      ;FOLD -- Start StartAcknowledge AUS -- ;%{SE}%MKUKATPVW %CVW_COM %VCOMMENT %P 2:-- Start StartAcknowledge AUS --, 3: VW_COMMENT
      ;ENDFOLD
      ;FOLD A3512 = AUS ;%{SE}%MKUKATPVW %CVW_SPS %VBOASG %P 2:A3512 = AUS, 3: BOASG
         $OUT[3512] = FALSE
      ;ENDFOLD
      ;FOLD -- RSK Fehlerausgabe Kraftaufbau -- ;%{SE}%MKUKATPVW %CVW_COM %VCOMMENT %P 2:-- RSK Fehlerausgabe Kraftaufbau --, 3: VW_COMMENT
      ;ENDFOLD
      ;FOLD F325 = EIN ;%{SE}%MKUKATPVW %CVW_SPS %VBOASG %P 2:F325 = EIN, 3: BOASG
         $FLAG[325] = TRUE
      ;ENDFOLD
      ;FOLD -- RSK Fehlerausgabe -- ;%{SE}%MKUKATPVW %CVW_COM %VCOMMENT %P 2:-- RSK Fehlerausgabe --, 3: VW_COMMENT
      ;ENDFOLD
      ;FOLD F327 = EIN ;%{SE}%MKUKATPVW %CVW_SPS %VBOASG %P 2:F327 = EIN, 3: BOASG
         $FLAG[327] = TRUE
      ;ENDFOLD
      ;FOLD F174 = !F327 & F174 ;%{SE}%MKUKATPVW %CVW_SPS %VBOASG %P 2:F174 = !F327 & F174, 3: BOASG
         $FLAG[174] = NOT $FLAG[327] AND $FLAG[174]
      ;ENDFOLD
      ;FOLD F175 = F327 + F175 ;%{SE}%MKUKATPVW %CVW_SPS %VBOASG %P 2:F175 = F327 + F175, 3: BOASG
         $FLAG[175] = $FLAG[327] OR $FLAG[175]
      ;ENDFOLD
      ;FOLD -- RSK Sammelstoerung -- ;%{SE}%MKUKATPVW %CVW_COM %VCOMMENT %P 2:-- RSK Sammelstoerung --, 3: VW_COMMENT
      ;ENDFOLD
      ;FOLD F329 = F325 + F326 + F327 ;%{SE}%MKUKATPVW %CVW_SPS %VBOASG %P 2:F329 = F325 + F326 + F327, 3: BOASG
         $FLAG[329] = $FLAG[325] OR $FLAG[326] OR $FLAG[327]
      ;ENDFOLD
      ;FOLD A3519 = EIN ;%{SE}%MKUKATPVW %CVW_SPS %VBOASG %P 2:A3519 = EIN, 3: BOASG
         $OUT[3519] = TRUE
      ;ENDFOLD
      ;FOLD -- Flagbildung Wiederholfraesen -- ;%{SE}%MKUKATPVW %CVW_COM %VCOMMENT %P 2:-- Flagbildung Wiederholfraesen --, 3: VW_COMMENT
      ;ENDFOLD
      ;FOLD F749 = F329 & !A3518 ;%{SE}%MKUKATPVW %CVW_SPS %VBOASG %P 2:F749 = F329 & !A3518, 3: BOASG
         $FLAG[749] = $FLAG[329] AND NOT $OUT[3518]
      ;ENDFOLD
      ;FOLD A204 = A3518 ;%{SE}%MKUKATPVW %CVW_SPS %VBOASG %P 2:A204 = A3518, 3: BOASG
         $OUT[204] = $OUT[3518]
      ;ENDFOLD
      ;FOLD Schritt 303 = A3926 & A3518 & (E26 + E27) ;%{SE}%MKUKATPVW %CVW_SPS %VST_CON %P 2:Schritt 303 = A3926 & A3518 & (E26 + E27), 3: ST_CON
         IF $OUT[3926] AND $OUT[3518] AND ($IN[26] OR $IN[27]) THEN
            PREV_STEP[9] = APP_INT_STEP[9]
            APP_INT_STEP[9] = 303
         ENDIF
      ;ENDFOLD
      ;FOLD Schritt 303 = A3926 & !A3518 & F749 & A4039 ;%{SE}%MKUKATPVW %CVW_SPS %VST_CON %P 2:Schritt 303 = A3926 & !A3518 & F749 & A4039, 3: ST_CON
         IF $OUT[3926] AND NOT $OUT[3518] AND $FLAG[749] AND $OUT[4039] THEN
            PREV_STEP[9] = APP_INT_STEP[9]
            APP_INT_STEP[9] = 303
         ENDIF
      ;ENDFOLD
   ;ENDFOLD
   ;FOLD SCHRITT 333 -- st. RZ3 # Acknowledge -- ;%{P}%MKUKATPVW,%CSTEP,%VST_NR,%P 1:SCHRITT, 2:333, 3: st. RZ3 # Acknowledge
      ;FOLD ;%{H}
         Case 333
      ;ENDFOLD
      ;FOLD -- ServoGun SZ1 oeffnen -- ;%{SE}%MKUKATPVW %CVW_COM %VCOMMENT %P 2:-- ServoGun SZ1 oeffnen --, 3: VW_COMMENT
      ;ENDFOLD
      ;FOLD A3511 = AUS ;%{SE}%MKUKATPVW %CVW_SPS %VBOASG %P 2:A3511 = AUS, 3: BOASG
         $OUT[3511] = FALSE
      ;ENDFOLD
      ;FOLD A3512 = EIN ;%{SE}%MKUKATPVW %CVW_SPS %VBOASG %P 2:A3512 = EIN, 3: BOASG
         $OUT[3512] = TRUE
      ;ENDFOLD
      ;FOLD -- RSK Fehlerausgabe Kraftaufbau -- ;%{SE}%MKUKATPVW %CVW_COM %VCOMMENT %P 2:-- RSK Fehlerausgabe Kraftaufbau --, 3: VW_COMMENT
      ;ENDFOLD
      ;FOLD F325 = AUS ;%{SE}%MKUKATPVW %CVW_SPS %VBOASG %P 2:F325 = AUS, 3: BOASG
         $FLAG[325] = FALSE
      ;ENDFOLD
      ;FOLD -- RSK Fehlerausgabe -- ;%{SE}%MKUKATPVW %CVW_COM %VCOMMENT %P 2:-- RSK Fehlerausgabe --, 3: VW_COMMENT
      ;ENDFOLD
      ;FOLD F327 = AUS ;%{SE}%MKUKATPVW %CVW_SPS %VBOASG %P 2:F327 = AUS, 3: BOASG
         $FLAG[327] = FALSE
      ;ENDFOLD
      ;FOLD -- RSK Fehlerausgabe -- ;%{SE}%MKUKATPVW %CVW_COM %VCOMMENT %P 2:-- RSK Fehlerausgabe --, 3: VW_COMMENT
      ;ENDFOLD
      ;FOLD F329 = AUS ;%{SE}%MKUKATPVW %CVW_SPS %VBOASG %P 2:F329 = AUS, 3: BOASG
         $FLAG[329] = FALSE
      ;ENDFOLD
      ;FOLD Schritt 334 = A3926 & A3506 & A3505 & !A3507 & A4039 ;%{SE}%MKUKATPVW %CVW_SPS %VST_CON %P 2:Schritt 334 = A3926 & A3506 & A3505 & !A3507 & A4039, 3: ST_CON
         IF $OUT[3926] AND $OUT[3506] AND $OUT[3505] AND NOT $OUT[3507] AND $OUT[4039] THEN
            PREV_STEP[9] = APP_INT_STEP[9]
            APP_INT_STEP[9] = 334
         ENDIF
      ;ENDFOLD
   ;ENDFOLD
   ;FOLD SCHRITT 334 -- st. RZ3 # Ende -- ;%{P}%MKUKATPVW,%CSTEP,%VST_NR,%P 1:SCHRITT, 2:334, 3: st. RZ3 # Ende
      ;FOLD ;%{H}
         Case 334
      ;ENDFOLD
      ;FOLD -- Hilfsflag SK Programmwechsel -- ;%{SE}%MKUKATPVW %CVW_COM %VCOMMENT %P 2:-- Hilfsflag SK Programmwechsel --, 3: VW_COMMENT
      ;ENDFOLD
      ;FOLD F334 = AUS ;%{SE}%MKUKATPVW %CVW_SPS %VBOASG %P 2:F334 = AUS, 3: BOASG
         $FLAG[334] = FALSE
      ;ENDFOLD
      ;FOLD A116 = AUS ;%{SE}%MKUKATPVW %CVW_SPS %VBOASG %P 2:A116 = AUS, 3: BOASG
         $OUT[116] = FALSE
      ;ENDFOLD
      ;FOLD A192 = AUS ;%{SE}%MKUKATPVW %CVW_SPS %VBOASG %P 2:A192 = AUS, 3: BOASG
         $OUT[192] = FALSE
      ;ENDFOLD
      ;FOLD A1107 = AUS ;%{SE}%MKUKATPVW %CVW_SPS %VBOASG %P 2:A1107 = AUS, 3: BOASG
         $OUT[1107] = FALSE
      ;ENDFOLD
      ;FOLD A3518 = AUS ;%{SE}%MKUKATPVW %CVW_SPS %VBOASG %P 2:A3518 = AUS, 3: BOASG
         $OUT[3518] = FALSE
      ;ENDFOLD
      ;FOLD A3519 = AUS ;%{SE}%MKUKATPVW %CVW_SPS %VBOASG %P 2:A3519 = AUS, 3: BOASG
         $OUT[3519] = FALSE
      ;ENDFOLD
      ;FOLD F836 = AUS ;%{SE}%MKUKATPVW %CVW_SPS %VBOASG %P 2:F836 = AUS, 3: BOASG
         $FLAG[836] = FALSE
      ;ENDFOLD
      ;FOLD -- Start Init Same AUS -- ;%{SE}%MKUKATPVW %CVW_COM %VCOMMENT %P 2:-- Start Init Same AUS --, 3: VW_COMMENT
      ;ENDFOLD
      ;FOLD A3514 = AUS ;%{SE}%MKUKATPVW %CVW_SPS %VBOASG %P 2:A3514 = AUS, 3: BOASG
         $OUT[3514] = FALSE
      ;ENDFOLD
      ;FOLD -- Start Spot AUS -- ;%{SE}%MKUKATPVW %CVW_COM %VCOMMENT %P 2:-- Start Spot AUS --, 3: VW_COMMENT
      ;ENDFOLD
      ;FOLD A3511 = AUS ;%{SE}%MKUKATPVW %CVW_SPS %VBOASG %P 2:A3511 = AUS, 3: BOASG
         $OUT[3511] = FALSE
      ;ENDFOLD
      ;FOLD -- Start Dress AUS -- ;%{SE}%MKUKATPVW %CVW_COM %VCOMMENT %P 2:-- Start Dress AUS --, 3: VW_COMMENT
      ;ENDFOLD
      ;FOLD A3510 = AUS ;%{SE}%MKUKATPVW %CVW_SPS %VBOASG %P 2:A3510 = AUS, 3: BOASG
         $OUT[3510] = FALSE
      ;ENDFOLD
      ;FOLD -- Start Init New AUS -- ;%{SE}%MKUKATPVW %CVW_COM %VCOMMENT %P 2:-- Start Init New AUS --, 3: VW_COMMENT
      ;ENDFOLD
      ;FOLD A3513 = AUS ;%{SE}%MKUKATPVW %CVW_SPS %VBOASG %P 2:A3513 = AUS, 3: BOASG
         $OUT[3513] = FALSE
      ;ENDFOLD
      ;FOLD -- Dress in Position AUS -- ;%{SE}%MKUKATPVW %CVW_COM %VCOMMENT %P 2:-- Dress in Position AUS --, 3: VW_COMMENT
      ;ENDFOLD
      ;FOLD A3935 = AUS ;%{SE}%MKUKATPVW %CVW_SPS %VBOASG %P 2:A3935 = AUS, 3: BOASG
         $OUT[3935] = FALSE
      ;ENDFOLD
      ;FOLD -- Dress Fin AUS -- ;%{SE}%MKUKATPVW %CVW_COM %VCOMMENT %P 2:-- Dress Fin AUS --, 3: VW_COMMENT
      ;ENDFOLD
      ;FOLD A3936 = AUS ;%{SE}%MKUKATPVW %CVW_SPS %VBOASG %P 2:A3936 = AUS, 3: BOASG
         $OUT[3936] = FALSE
      ;ENDFOLD
      ;FOLD -- Start StartAcknowledge AUS -- ;%{SE}%MKUKATPVW %CVW_COM %VCOMMENT %P 2:-- Start StartAcknowledge AUS --, 3: VW_COMMENT
      ;ENDFOLD
      ;FOLD A3512 = AUS ;%{SE}%MKUKATPVW %CVW_SPS %VBOASG %P 2:A3512 = AUS, 3: BOASG
         $OUT[3512] = FALSE
      ;ENDFOLD
      ;FOLD -- RSK Sammelstoerung -- ;%{SE}%MKUKATPVW %CVW_COM %VCOMMENT %P 2:-- RSK Sammelstoerung --, 3: VW_COMMENT
      ;ENDFOLD
      ;FOLD F329 = F196 ;%{SE}%MKUKATPVW %CVW_SPS %VBOASG %P 2:F329 = F196, 3: BOASG
         $FLAG[329] = $FLAG[196]
      ;ENDFOLD
      ;FOLD F185 = (!E1106 & E787 & !E1108 & !F830) + F196 & (E26 + E27) ;%{SE}%MKUKATPVW %CVW_SPS %VBOASG %P 2:F185 = (!E1106 & E787 & !E1108 & !F830) + F196 & (E26 + E27), 3: BOASG
         $FLAG[185] = (NOT $IN[1106] AND $IN[787] AND NOT $IN[1108] AND NOT $FLAG[830]) OR $FLAG[196] AND ($IN[26] OR $IN[27])
      ;ENDFOLD
      ;FOLD SCHRITT 1 = F185 & A4039 & A3926 & A3506 & A3505 ;%{SE}%MKUKATPVW %CVW_SPS %VST_CON %P 2:SCHRITT 1 = F185 & A4039 & A3926 & A3506 & A3505, 3: ST_CON
         IF $FLAG[185] AND $OUT[4039] AND $OUT[3926] AND $OUT[3506] AND $OUT[3505] THEN
            PREV_STEP[9] = APP_INT_STEP[9]
            APP_INT_STEP[9] = 1
         ENDIF
      ;ENDFOLD
   ;ENDFOLD
   ;FOLD SCHRITT 350 -- st. RZ3 # Fehler SGB -- ;%{P}%MKUKATPVW,%CSTEP,%VST_NR,%P 1:SCHRITT, 2:350, 3: st. RZ3 # Fehler SGB
      ;FOLD ;%{H}
         Case 350
      ;ENDFOLD
      ;FOLD -- Start Init Same AUS -- ;%{SE}%MKUKATPVW %CVW_COM %VCOMMENT %P 2:-- Start Init Same AUS --, 3: VW_COMMENT
      ;ENDFOLD
      ;FOLD A3514 = AUS ;%{SE}%MKUKATPVW %CVW_SPS %VBOASG %P 2:A3514 = AUS, 3: BOASG
         $OUT[3514] = FALSE
      ;ENDFOLD
      ;FOLD -- Start Spot AUS -- ;%{SE}%MKUKATPVW %CVW_COM %VCOMMENT %P 2:-- Start Spot AUS --, 3: VW_COMMENT
      ;ENDFOLD
      ;FOLD A3511 = AUS ;%{SE}%MKUKATPVW %CVW_SPS %VBOASG %P 2:A3511 = AUS, 3: BOASG
         $OUT[3511] = FALSE
      ;ENDFOLD
      ;FOLD -- Start Dress AUS -- ;%{SE}%MKUKATPVW %CVW_COM %VCOMMENT %P 2:-- Start Dress AUS --, 3: VW_COMMENT
      ;ENDFOLD
      ;FOLD A3510 = AUS ;%{SE}%MKUKATPVW %CVW_SPS %VBOASG %P 2:A3510 = AUS, 3: BOASG
         $OUT[3510] = FALSE
      ;ENDFOLD
      ;FOLD -- Start Init New AUS -- ;%{SE}%MKUKATPVW %CVW_COM %VCOMMENT %P 2:-- Start Init New AUS --, 3: VW_COMMENT
      ;ENDFOLD
      ;FOLD A3513 = AUS ;%{SE}%MKUKATPVW %CVW_SPS %VBOASG %P 2:A3513 = AUS, 3: BOASG
         $OUT[3513] = FALSE
      ;ENDFOLD
      ;FOLD -- Start Dress in Position AUS -- ;%{SE}%MKUKATPVW %CVW_COM %VCOMMENT %P 2:-- Start Dress in Position AUS --, 3: VW_COMMENT
      ;ENDFOLD
      ;FOLD A3935 = AUS ;%{SE}%MKUKATPVW %CVW_SPS %VBOASG %P 2:A3935 = AUS, 3: BOASG
         $OUT[3935] = FALSE
      ;ENDFOLD
      ;FOLD -- Start Dress Fin AUS -- ;%{SE}%MKUKATPVW %CVW_COM %VCOMMENT %P 2:-- Start Dress Fin AUS --, 3: VW_COMMENT
      ;ENDFOLD
      ;FOLD A3936 = AUS ;%{SE}%MKUKATPVW %CVW_SPS %VBOASG %P 2:A3936 = AUS, 3: BOASG
         $OUT[3936] = FALSE
      ;ENDFOLD
      ;FOLD -- Start StartAcknowledge EIN -- ;%{SE}%MKUKATPVW %CVW_COM %VCOMMENT %P 2:-- Start StartAcknowledge EIN --, 3: VW_COMMENT
      ;ENDFOLD
      ;FOLD A3512 = EIN ;%{SE}%MKUKATPVW %CVW_SPS %VBOASG %P 2:A3512 = EIN, 3: BOASG
         $OUT[3512] = TRUE
      ;ENDFOLD
      ;FOLD -- Kommentar -- ;%{SE}%MKUKATPVW %CVW_COM %VCOMMENT %P 2:-- Kommentar --, 3: VW_COMMENT
      ;ENDFOLD
      ;FOLD Schritt 351 = A4039 & A140 & !A3507 & A3506 & A3505 ;%{SE}%MKUKATPVW %CVW_SPS %VST_CON %P 2:Schritt 351 = A4039 & A140 & !A3507 & A3506 & A3505, 3: ST_CON
         IF $OUT[4039] AND $OUT[140] AND NOT $OUT[3507] AND $OUT[3506] AND $OUT[3505] THEN
            PREV_STEP[9] = APP_INT_STEP[9]
            APP_INT_STEP[9] = 351
         ENDIF
      ;ENDFOLD
   ;ENDFOLD
   ;FOLD SCHRITT 351 -- st. RZ3 # Fehler SGB -- ;%{P}%MKUKATPVW,%CSTEP,%VST_NR,%P 1:SCHRITT, 2:351, 3: st. RZ3 # Fehler SGB
      ;FOLD ;%{H}
         Case 351
      ;ENDFOLD
      ;FOLD -- Start StartAcknowledge AUS -- ;%{SE}%MKUKATPVW %CVW_COM %VCOMMENT %P 2:-- Start StartAcknowledge AUS --, 3: VW_COMMENT
      ;ENDFOLD
      ;FOLD A3512 = AUS ;%{SE}%MKUKATPVW %CVW_SPS %VBOASG %P 2:A3512 = AUS, 3: BOASG
         $OUT[3512] = FALSE
      ;ENDFOLD
      ;FOLD SCHRITT 1 = A4039 & A204 ;%{SE}%MKUKATPVW %CVW_SPS %VST_CON %P 2:SCHRITT 1 = A4039 & A204, 3: ST_CON
         IF $OUT[4039] AND $OUT[204] THEN
            PREV_STEP[9] = APP_INT_STEP[9]
            APP_INT_STEP[9] = 1
         ENDIF
      ;ENDFOLD
   ;ENDFOLD
   ;FOLD SCHRITT 390 -- st. RZ3 Setzhub 2 -- ;%{P}%MKUKATPVW,%CSTEP,%VST_NR,%P 1:SCHRITT, 2:390, 3: st. RZ3 Setzhub 2
      ;FOLD ;%{H}
         Case 390
      ;ENDFOLD
      ;FOLD -- Druckvorgabe SK1/ServoGun -- ;%{SE}%MKUKATPVW %CVW_COM %VCOMMENT %P 2:-- Druckvorgabe SK1/ServoGun --, 3: VW_COMMENT
      ;ENDFOLD
      ;FOLD bin7 ( F174 ) = 61 ;%{SE}%MKUKATPVW %CVW_SPS %VARIASG %P 2:bin7 ( F174 ) = 61, 3: ARIASG
         VW(#BINOUT,$FLAG[174],7,61)
      ;ENDFOLD
      ;FOLD bin31 ( F174 ) = 61 ;%{SE}%MKUKATPVW %CVW_SPS %VARIASG %P 2:bin31 ( F174 ) = 61, 3: ARIASG
         VW(#BINOUT,$FLAG[174],31,61)
      ;ENDFOLD
      ;FOLD -- Wartezeit Programmwechsel SK -- ;%{SE}%MKUKATPVW %CVW_COM %VCOMMENT %P 2:-- Wartezeit Programmwechsel SK --, 3: VW_COMMENT
      ;ENDFOLD
      ;FOLD T8 ( !F334 ) = -2[1/10Sek] ;%{SE}%MKUKATPVW %CVW_SPS %VTASG %P 2:T8 ( !F334 ) = -2[1/10Sek], 3: TASG
         VW(#SET_TIME,NOT $FLAG[334],8,0,-2)
      ;ENDFOLD
      ;FOLD -- Ueberwachungszeit ServoGun Setzhub 2 -- ;%{SE}%MKUKATPVW %CVW_COM %VCOMMENT %P 2:-- Ueberwachungszeit ServoGun Setzhub 2 --, 3: VW_COMMENT
      ;ENDFOLD
      ;FOLD t9 ( EIN ) = -80[1/10Sek] ;%{SE}%MKUKATPVW %CVW_SPS %VTASG %P 2:t9 ( EIN ) = -80[1/10Sek], 3: TASG
         VW(#SET_TIME,TRUE,9,0,-80)
      ;ENDFOLD
      ;FOLD -- Hilfsflag SK Programmwechsel -- ;%{SE}%MKUKATPVW %CVW_COM %VCOMMENT %P 2:-- Hilfsflag SK Programmwechsel --, 3: VW_COMMENT
      ;ENDFOLD
      ;FOLD F334 = EIN ;%{SE}%MKUKATPVW %CVW_SPS %VBOASG %P 2:F334 = EIN, 3: BOASG
         $FLAG[334] = TRUE
      ;ENDFOLD
      ;FOLD A3512 = AUS ;%{SE}%MKUKATPVW %CVW_SPS %VBOASG %P 2:A3512 = AUS, 3: BOASG
         $OUT[3512] = FALSE
      ;ENDFOLD
      ;FOLD Schritt 391 = T8 & A4039 & A3506 & A3505 & !A3507 ;%{SE}%MKUKATPVW %CVW_SPS %VST_CON %P 2:Schritt 391 = T8 & A4039 & A3506 & A3505 & !A3507, 3: ST_CON
         IF $TIMER_FLAG[8] AND $OUT[4039] AND $OUT[3506] AND $OUT[3505] AND NOT $OUT[3507] THEN
            PREV_STEP[9] = APP_INT_STEP[9]
            APP_INT_STEP[9] = 391
         ENDIF
      ;ENDFOLD
   ;ENDFOLD
   ;FOLD SCHRITT 391 -- st. RZ3 Setzhub 2 # InitSame -- ;%{P}%MKUKATPVW,%CSTEP,%VST_NR,%P 1:SCHRITT, 2:391, 3: st. RZ3 Setzhub 2 # InitSame
      ;FOLD ;%{H}
         Case 391
      ;ENDFOLD
      ;FOLD -- Hilfsflag SK Programmwechsel -- ;%{SE}%MKUKATPVW %CVW_COM %VCOMMENT %P 2:-- Hilfsflag SK Programmwechsel --, 3: VW_COMMENT
      ;ENDFOLD
      ;FOLD F334 = AUS ;%{SE}%MKUKATPVW %CVW_SPS %VBOASG %P 2:F334 = AUS, 3: BOASG
         $FLAG[334] = FALSE
      ;ENDFOLD
      ;FOLD -- Zeit fuer Setzhub -- ;%{SE}%MKUKATPVW %CVW_COM %VCOMMENT %P 2:-- Zeit fuer Setzhub --, 3: VW_COMMENT
      ;ENDFOLD
      ;FOLD T8 ( EIN ) = -80[1/10Sek] ;%{SE}%MKUKATPVW %CVW_SPS %VTASG %P 2:T8 ( EIN ) = -80[1/10Sek], 3: TASG
         VW(#SET_TIME,TRUE,8,0,-80)
      ;ENDFOLD
      ;FOLD -- Messen nach Fraesen -- ;%{SE}%MKUKATPVW %CVW_COM %VCOMMENT %P 2:-- Messen nach Fraesen --, 3: VW_COMMENT
      ;ENDFOLD
      ;FOLD A3514 = EIN ;%{SE}%MKUKATPVW %CVW_SPS %VBOASG %P 2:A3514 = EIN, 3: BOASG
         $OUT[3514] = TRUE
      ;ENDFOLD
      ;FOLD A3510 = EIN ;%{SE}%MKUKATPVW %CVW_SPS %VBOASG %P 2:A3510 = EIN, 3: BOASG
         $OUT[3510] = TRUE
      ;ENDFOLD
      ;FOLD Schritt 392 = A4039 ;%{SE}%MKUKATPVW %CVW_SPS %VST_CON %P 2:Schritt 392 = A4039, 3: ST_CON
         IF $OUT[4039] THEN
            PREV_STEP[9] = APP_INT_STEP[9]
            APP_INT_STEP[9] = 392
         ENDIF
      ;ENDFOLD
   ;ENDFOLD
   ;FOLD SCHRITT 392 -- st. RZ3 Setzhub 2 # Auswertung -- ;%{P}%MKUKATPVW,%CSTEP,%VST_NR,%P 1:SCHRITT, 2:392, 3: st. RZ3 Setzhub 2 # Auswertung
      ;FOLD ;%{H}
         Case 392
      ;ENDFOLD
      ;FOLD -- Hilfsflag SK Programmwechsel -- ;%{SE}%MKUKATPVW %CVW_COM %VCOMMENT %P 2:-- Hilfsflag SK Programmwechsel --, 3: VW_COMMENT
      ;ENDFOLD
      ;FOLD F334 = AUS ;%{SE}%MKUKATPVW %CVW_SPS %VBOASG %P 2:F334 = AUS, 3: BOASG
         $FLAG[334] = FALSE
      ;ENDFOLD
      ;FOLD -- Warte Ergebnis -- ;%{SE}%MKUKATPVW %CVW_COM %VCOMMENT %P 2:-- Warte Ergebnis --, 3: VW_COMMENT
      ;ENDFOLD
      ;FOLD Schritt 393 = A3508 & A4039 + T8 + T9 ;%{SE}%MKUKATPVW %CVW_SPS %VST_CON %P 2:Schritt 393 = A3508 & A4039 + T8 + T9, 3: ST_CON
         IF $OUT[3508] AND $OUT[4039] OR $TIMER_FLAG[8] OR $TIMER_FLAG[9] THEN
            PREV_STEP[9] = APP_INT_STEP[9]
            APP_INT_STEP[9] = 393
         ENDIF
      ;ENDFOLD
   ;ENDFOLD
   ;FOLD SCHRITT 393 -- st. RZ3 Setzhub 2 # Acknowledge -- ;%{P}%MKUKATPVW,%CSTEP,%VST_NR,%P 1:SCHRITT, 2:393, 3: st. RZ3 Setzhub 2 # Acknowledge
      ;FOLD ;%{H}
         Case 393
      ;ENDFOLD
      ;FOLD -- RSK Fehlerausgabe Kraftaufbau -- ;%{SE}%MKUKATPVW %CVW_COM %VCOMMENT %P 2:-- RSK Fehlerausgabe Kraftaufbau --, 3: VW_COMMENT
      ;ENDFOLD
      ;FOLD F325 = !A3508 & T9 ;%{SE}%MKUKATPVW %CVW_SPS %VBOASG %P 2:F325 = !A3508 & T9, 3: BOASG
         $FLAG[325] = NOT $OUT[3508] AND $TIMER_FLAG[9]
      ;ENDFOLD
      ;FOLD F329 = T9 ;%{SE}%MKUKATPVW %CVW_SPS %VBOASG %P 2:F329 = T9, 3: BOASG
         $FLAG[329] = $TIMER_FLAG[9]
      ;ENDFOLD
      ;FOLD -- ServoGun SZ1 oeffnen -- ;%{SE}%MKUKATPVW %CVW_COM %VCOMMENT %P 2:-- ServoGun SZ1 oeffnen --, 3: VW_COMMENT
      ;ENDFOLD
      ;FOLD -- RSK Fehlerausgabe Messen -- ;%{SE}%MKUKATPVW %CVW_COM %VCOMMENT %P 2:-- RSK Fehlerausgabe Messen --, 3: VW_COMMENT
      ;ENDFOLD
      ;FOLD A3510 = AUS ;%{SE}%MKUKATPVW %CVW_SPS %VBOASG %P 2:A3510 = AUS, 3: BOASG
         $OUT[3510] = FALSE
      ;ENDFOLD
      ;FOLD A3514 = AUS ;%{SE}%MKUKATPVW %CVW_SPS %VBOASG %P 2:A3514 = AUS, 3: BOASG
         $OUT[3514] = FALSE
      ;ENDFOLD
      ;FOLD A3512 = EIN ;%{SE}%MKUKATPVW %CVW_SPS %VBOASG %P 2:A3512 = EIN, 3: BOASG
         $OUT[3512] = TRUE
      ;ENDFOLD
      ;FOLD -- Druckvorgabe SK1/ServoGun -- ;%{SE}%MKUKATPVW %CVW_COM %VCOMMENT %P 2:-- Druckvorgabe SK1/ServoGun --, 3: VW_COMMENT
      ;ENDFOLD
      ;FOLD bin7 ( F174 ) = 41 ;%{SE}%MKUKATPVW %CVW_SPS %VARIASG %P 2:bin7 ( F174 ) = 41, 3: ARIASG
         VW(#BINOUT,$FLAG[174],7,41)
      ;ENDFOLD
      ;FOLD bin7 ( F175 ) = 51 ;%{SE}%MKUKATPVW %CVW_SPS %VARIASG %P 2:bin7 ( F175 ) = 51, 3: ARIASG
         VW(#BINOUT,$FLAG[175],7,51)
      ;ENDFOLD
      ;FOLD bin31 ( F174 ) = 41 ;%{SE}%MKUKATPVW %CVW_SPS %VARIASG %P 2:bin31 ( F174 ) = 41, 3: ARIASG
         VW(#BINOUT,$FLAG[174],31,41)
      ;ENDFOLD
      ;FOLD bin31 ( F175 ) = 51 ;%{SE}%MKUKATPVW %CVW_SPS %VARIASG %P 2:bin31 ( F175 ) = 51, 3: ARIASG
         VW(#BINOUT,$FLAG[175],31,51)
      ;ENDFOLD
      ;FOLD -- Wartezeit Programmwechsel SK -- ;%{SE}%MKUKATPVW %CVW_COM %VCOMMENT %P 2:-- Wartezeit Programmwechsel SK --, 3: VW_COMMENT
      ;ENDFOLD
      ;FOLD T8 ( !F334 ) = -2[1/10Sek] ;%{SE}%MKUKATPVW %CVW_SPS %VTASG %P 2:T8 ( !F334 ) = -2[1/10Sek], 3: TASG
         VW(#SET_TIME,NOT $FLAG[334],8,0,-2)
      ;ENDFOLD
      ;FOLD -- Hilfsflag SK Programmwechsel -- ;%{SE}%MKUKATPVW %CVW_COM %VCOMMENT %P 2:-- Hilfsflag SK Programmwechsel --, 3: VW_COMMENT
      ;ENDFOLD
      ;FOLD F334 = EIN ;%{SE}%MKUKATPVW %CVW_SPS %VBOASG %P 2:F334 = EIN, 3: BOASG
         $FLAG[334] = TRUE
      ;ENDFOLD
      ;FOLD Schritt 394 = T8 & A4039 & !A3507 ;%{SE}%MKUKATPVW %CVW_SPS %VST_CON %P 2:Schritt 394 = T8 & A4039 & !A3507, 3: ST_CON
         IF $TIMER_FLAG[8] AND $OUT[4039] AND NOT $OUT[3507] THEN
            PREV_STEP[9] = APP_INT_STEP[9]
            APP_INT_STEP[9] = 394
         ENDIF
      ;ENDFOLD
   ;ENDFOLD
   ;FOLD SCHRITT 394 -- st. RZ3 Setzhub 2 -- ;%{P}%MKUKATPVW,%CSTEP,%VST_NR,%P 1:SCHRITT, 2:394, 3: st. RZ3 Setzhub 2
      ;FOLD ;%{H}
         Case 394
      ;ENDFOLD
      ;FOLD -- Hilfsflag SK Programmwechsel -- ;%{SE}%MKUKATPVW %CVW_COM %VCOMMENT %P 2:-- Hilfsflag SK Programmwechsel --, 3: VW_COMMENT
      ;ENDFOLD
      ;FOLD F334 = AUS ;%{SE}%MKUKATPVW %CVW_SPS %VBOASG %P 2:F334 = AUS, 3: BOASG
         $FLAG[334] = FALSE
      ;ENDFOLD
      ;FOLD A3512 = AUS ;%{SE}%MKUKATPVW %CVW_SPS %VBOASG %P 2:A3512 = AUS, 3: BOASG
         $OUT[3512] = FALSE
      ;ENDFOLD
      ;FOLD Schritt 329 = A4039  & A3506 & A3505 & !A3507 ;%{SE}%MKUKATPVW %CVW_SPS %VST_CON %P 2:Schritt 329 = A4039  & A3506 & A3505 & !A3507, 3: ST_CON
         IF $OUT[4039] AND $OUT[3506] AND $OUT[3505] AND NOT $OUT[3507] THEN
            PREV_STEP[9] = APP_INT_STEP[9]
            APP_INT_STEP[9] = 329
         ENDIF
      ;ENDFOLD
   ;ENDFOLD
   ;FOLD SCHRITT 500 -- rob. RZ # Ruecksetzen -- ;%{P}%MKUKATPVW,%CSTEP,%VST_NR,%P 1:SCHRITT, 2:500, 3: rob. RZ # Ruecksetzen
      ;FOLD ;%{H}
         Case 500
      ;ENDFOLD
      ;FOLD -- Schrittkette gestartet -- ;%{SE}%MKUKATPVW %CVW_COM %VCOMMENT %P 2:-- Schrittkette gestartet --, 3: VW_COMMENT
      ;ENDFOLD
      ;FOLD F276 = EIN ;%{SE}%MKUKATPVW %CVW_SPS %VBOASG %P 2:F276 = EIN, 3: BOASG
         $FLAG[276] = TRUE
      ;ENDFOLD
      ;FOLD -- Start Init Same AUS -- ;%{SE}%MKUKATPVW %CVW_COM %VCOMMENT %P 2:-- Start Init Same AUS --, 3: VW_COMMENT
      ;ENDFOLD
      ;FOLD A3514 = AUS ;%{SE}%MKUKATPVW %CVW_SPS %VBOASG %P 2:A3514 = AUS, 3: BOASG
         $OUT[3514] = FALSE
      ;ENDFOLD
      ;FOLD -- Start Spot AUS -- ;%{SE}%MKUKATPVW %CVW_COM %VCOMMENT %P 2:-- Start Spot AUS --, 3: VW_COMMENT
      ;ENDFOLD
      ;FOLD A3511 = AUS ;%{SE}%MKUKATPVW %CVW_SPS %VBOASG %P 2:A3511 = AUS, 3: BOASG
         $OUT[3511] = FALSE
      ;ENDFOLD
      ;FOLD -- Start Dress AUS -- ;%{SE}%MKUKATPVW %CVW_COM %VCOMMENT %P 2:-- Start Dress AUS --, 3: VW_COMMENT
      ;ENDFOLD
      ;FOLD A3510 = AUS ;%{SE}%MKUKATPVW %CVW_SPS %VBOASG %P 2:A3510 = AUS, 3: BOASG
         $OUT[3510] = FALSE
      ;ENDFOLD
      ;FOLD -- Start Init New AUS -- ;%{SE}%MKUKATPVW %CVW_COM %VCOMMENT %P 2:-- Start Init New AUS --, 3: VW_COMMENT
      ;ENDFOLD
      ;FOLD A3513 = AUS ;%{SE}%MKUKATPVW %CVW_SPS %VBOASG %P 2:A3513 = AUS, 3: BOASG
         $OUT[3513] = FALSE
      ;ENDFOLD
      ;FOLD -- Start Dress in Position AUS -- ;%{SE}%MKUKATPVW %CVW_COM %VCOMMENT %P 2:-- Start Dress in Position AUS --, 3: VW_COMMENT
      ;ENDFOLD
      ;FOLD A3935 = AUS ;%{SE}%MKUKATPVW %CVW_SPS %VBOASG %P 2:A3935 = AUS, 3: BOASG
         $OUT[3935] = FALSE
      ;ENDFOLD
      ;FOLD -- Start Dress Fin AUS -- ;%{SE}%MKUKATPVW %CVW_COM %VCOMMENT %P 2:-- Start Dress Fin AUS --, 3: VW_COMMENT
      ;ENDFOLD
      ;FOLD A3936 = AUS ;%{SE}%MKUKATPVW %CVW_SPS %VBOASG %P 2:A3936 = AUS, 3: BOASG
         $OUT[3936] = FALSE
      ;ENDFOLD
      ;FOLD -- Start StartAcknowledge AUS -- ;%{SE}%MKUKATPVW %CVW_COM %VCOMMENT %P 2:-- Start StartAcknowledge AUS --, 3: VW_COMMENT
      ;ENDFOLD
      ;FOLD A3512 = AUS ;%{SE}%MKUKATPVW %CVW_SPS %VBOASG %P 2:A3512 = AUS, 3: BOASG
         $OUT[3512] = FALSE
      ;ENDFOLD
      ;FOLD -- Fehler SK ruecksetzen -- ;%{SE}%MKUKATPVW %CVW_COM %VCOMMENT %P 2:-- Fehler SK ruecksetzen --, 3: VW_COMMENT
      ;ENDFOLD
      ;FOLD -- Fehler SK Messen AUS -- ;%{SE}%MKUKATPVW %CVW_COM %VCOMMENT %P 2:-- Fehler SK Messen AUS --, 3: VW_COMMENT
      ;ENDFOLD
      ;FOLD F326 = AUS ;%{SE}%MKUKATPVW %CVW_SPS %VBOASG %P 2:F326 = AUS, 3: BOASG
         $FLAG[326] = FALSE
      ;ENDFOLD
      ;FOLD -- Fehler SK Gesamt AUS -- ;%{SE}%MKUKATPVW %CVW_COM %VCOMMENT %P 2:-- Fehler SK Gesamt AUS --, 3: VW_COMMENT
      ;ENDFOLD
      ;FOLD F326 = AUS ;%{SE}%MKUKATPVW %CVW_SPS %VBOASG %P 2:F326 = AUS, 3: BOASG
         $FLAG[326] = FALSE
      ;ENDFOLD
      ;FOLD Schritt 501 = A4039 & A3506 & A3505 & !E838 ;%{SE}%MKUKATPVW %CVW_SPS %VST_CON %P 2:Schritt 501 = A4039 & A3506 & A3505 & !E838, 3: ST_CON
         IF $OUT[4039] AND $OUT[3506] AND $OUT[3505] AND NOT $IN[838] THEN
            PREV_STEP[9] = APP_INT_STEP[9]
            APP_INT_STEP[9] = 501
         ENDIF
      ;ENDFOLD
   ;ENDFOLD
   ;FOLD SCHRITT 501 -- rob. RZ # Init Same -- ;%{P}%MKUKATPVW,%CSTEP,%VST_NR,%P 1:SCHRITT, 2:501, 3: rob. RZ # Init Same
      ;FOLD ;%{H}
         Case 501
      ;ENDFOLD
      ;FOLD -- Messen nach Fraesen -- ;%{SE}%MKUKATPVW %CVW_COM %VCOMMENT %P 2:-- Messen nach Fraesen --, 3: VW_COMMENT
      ;ENDFOLD
      ;FOLD -- Start Init Same AUS -- ;%{SE}%MKUKATPVW %CVW_COM %VCOMMENT %P 2:-- Start Init Same AUS --, 3: VW_COMMENT
      ;ENDFOLD
      ;FOLD A3514 = A3506 & A3505 ;%{SE}%MKUKATPVW %CVW_SPS %VBOASG %P 2:A3514 = A3506 & A3505, 3: BOASG
         $OUT[3514] = $OUT[3506] AND $OUT[3505]
      ;ENDFOLD
      ;FOLD -- Start Dress wenn Hintergrund bereit -- ;%{SE}%MKUKATPVW %CVW_COM %VCOMMENT %P 2:-- Start Dress wenn Hintergrund bereit --, 3: VW_COMMENT
      ;ENDFOLD
      ;FOLD A3510 = A3506 & A3505 ;%{SE}%MKUKATPVW %CVW_SPS %VBOASG %P 2:A3510 = A3506 & A3505, 3: BOASG
         $OUT[3510] = $OUT[3506] AND $OUT[3505]
      ;ENDFOLD
      ;FOLD Schritt 502 = A4039 & A3507 ;%{SE}%MKUKATPVW %CVW_SPS %VST_CON %P 2:Schritt 502 = A4039 & A3507, 3: ST_CON
         IF $OUT[4039] AND $OUT[3507] THEN
            PREV_STEP[9] = APP_INT_STEP[9]
            APP_INT_STEP[9] = 502
         ENDIF
      ;ENDFOLD
   ;ENDFOLD
   ;FOLD SCHRITT 502 -- rob. RZ # Anwahl -- ;%{P}%MKUKATPVW,%CSTEP,%VST_NR,%P 1:SCHRITT, 2:502, 3: rob. RZ # Anwahl
      ;FOLD ;%{H}
         Case 502
      ;ENDFOLD
      ;FOLD -- Fraeser ausblasen -- ;%{SE}%MKUKATPVW %CVW_COM %VCOMMENT %P 2:-- Fraeser ausblasen --, 3: VW_COMMENT
      ;ENDFOLD
      ;FOLD A834 = !F749 ;%{SE}%MKUKATPVW %CVW_SPS %VBOASG %P 2:A834 = !F749, 3: BOASG
         $OUT[834] = NOT $FLAG[749]
      ;ENDFOLD
      ;FOLD A835 = !F749 ;%{SE}%MKUKATPVW %CVW_SPS %VBOASG %P 2:A835 = !F749, 3: BOASG
         $OUT[835] = NOT $FLAG[749]
      ;ENDFOLD
      ;FOLD A858 = F289 ;%{SE}%MKUKATPVW %CVW_SPS %VBOASG %P 2:A858 = F289, 3: BOASG
         $OUT[858] = $FLAG[289]
      ;ENDFOLD
      ;FOLD A859 = F289 ;%{SE}%MKUKATPVW %CVW_SPS %VBOASG %P 2:A859 = F289, 3: BOASG
         $OUT[859] = $FLAG[289]
      ;ENDFOLD
      ;FOLD Schritt 503 = A4039 ;%{SE}%MKUKATPVW %CVW_SPS %VST_CON %P 2:Schritt 503 = A4039, 3: ST_CON
         IF $OUT[4039] THEN
            PREV_STEP[9] = APP_INT_STEP[9]
            APP_INT_STEP[9] = 503
         ENDIF
      ;ENDFOLD
   ;ENDFOLD
   ;FOLD SCHRITT 503 -- rob. RZ # Auswertung -- ;%{P}%MKUKATPVW,%CSTEP,%VST_NR,%P 1:SCHRITT, 2:503, 3: rob. RZ # Auswertung
      ;FOLD ;%{H}
         Case 503
      ;ENDFOLD
      ;FOLD -- Auswertung -- ;%{SE}%MKUKATPVW %CVW_COM %VCOMMENT %P 2:-- Auswertung --, 3: VW_COMMENT
      ;ENDFOLD
      ;FOLD Schritt 505 = A4039 & A3508 ;%{SE}%MKUKATPVW %CVW_SPS %VST_CON %P 2:Schritt 505 = A4039 & A3508, 3: ST_CON
         IF $OUT[4039] AND $OUT[3508] THEN
            PREV_STEP[9] = APP_INT_STEP[9]
            APP_INT_STEP[9] = 505
         ENDIF
      ;ENDFOLD
      ;FOLD Schritt 504 = A4039 & A3509 ;%{SE}%MKUKATPVW %CVW_SPS %VST_CON %P 2:Schritt 504 = A4039 & A3509, 3: ST_CON
         IF $OUT[4039] AND $OUT[3509] THEN
            PREV_STEP[9] = APP_INT_STEP[9]
            APP_INT_STEP[9] = 504
         ENDIF
      ;ENDFOLD
   ;ENDFOLD
   ;FOLD SCHRITT 504 -- rob. RZ # Fehlerfall -- ;%{P}%MKUKATPVW,%CSTEP,%VST_NR,%P 1:SCHRITT, 2:504, 3: rob. RZ # Fehlerfall
      ;FOLD ;%{H}
         Case 504
      ;ENDFOLD
      ;FOLD -- Ausblasen AUS -- ;%{SE}%MKUKATPVW %CVW_COM %VCOMMENT %P 2:-- Ausblasen AUS --, 3: VW_COMMENT
      ;ENDFOLD
      ;FOLD A834 = AUS ;%{SE}%MKUKATPVW %CVW_SPS %VBOASG %P 2:A834 = AUS, 3: BOASG
         $OUT[834] = FALSE
      ;ENDFOLD
      ;FOLD A835 = AUS ;%{SE}%MKUKATPVW %CVW_SPS %VBOASG %P 2:A835 = AUS, 3: BOASG
         $OUT[835] = FALSE
      ;ENDFOLD
      ;FOLD A858 = AUS ;%{SE}%MKUKATPVW %CVW_SPS %VBOASG %P 2:A858 = AUS, 3: BOASG
         $OUT[858] = FALSE
      ;ENDFOLD
      ;FOLD A859 = AUS ;%{SE}%MKUKATPVW %CVW_SPS %VBOASG %P 2:A859 = AUS, 3: BOASG
         $OUT[859] = FALSE
      ;ENDFOLD
      ;FOLD -- Start Init Same AUS -- ;%{SE}%MKUKATPVW %CVW_COM %VCOMMENT %P 2:-- Start Init Same AUS --, 3: VW_COMMENT
      ;ENDFOLD
      ;FOLD A3514 = AUS ;%{SE}%MKUKATPVW %CVW_SPS %VBOASG %P 2:A3514 = AUS, 3: BOASG
         $OUT[3514] = FALSE
      ;ENDFOLD
      ;FOLD -- Start Spot AUS -- ;%{SE}%MKUKATPVW %CVW_COM %VCOMMENT %P 2:-- Start Spot AUS --, 3: VW_COMMENT
      ;ENDFOLD
      ;FOLD A3511 = AUS ;%{SE}%MKUKATPVW %CVW_SPS %VBOASG %P 2:A3511 = AUS, 3: BOASG
         $OUT[3511] = FALSE
      ;ENDFOLD
      ;FOLD -- Start Dress AUS -- ;%{SE}%MKUKATPVW %CVW_COM %VCOMMENT %P 2:-- Start Dress AUS --, 3: VW_COMMENT
      ;ENDFOLD
      ;FOLD A3510 = AUS ;%{SE}%MKUKATPVW %CVW_SPS %VBOASG %P 2:A3510 = AUS, 3: BOASG
         $OUT[3510] = FALSE
      ;ENDFOLD
      ;FOLD -- Start Init New AUS -- ;%{SE}%MKUKATPVW %CVW_COM %VCOMMENT %P 2:-- Start Init New AUS --, 3: VW_COMMENT
      ;ENDFOLD
      ;FOLD A3513 = AUS ;%{SE}%MKUKATPVW %CVW_SPS %VBOASG %P 2:A3513 = AUS, 3: BOASG
         $OUT[3513] = FALSE
      ;ENDFOLD
      ;FOLD -- Start Dress in Position AUS -- ;%{SE}%MKUKATPVW %CVW_COM %VCOMMENT %P 2:-- Start Dress in Position AUS --, 3: VW_COMMENT
      ;ENDFOLD
      ;FOLD A3935 = AUS ;%{SE}%MKUKATPVW %CVW_SPS %VBOASG %P 2:A3935 = AUS, 3: BOASG
         $OUT[3935] = FALSE
      ;ENDFOLD
      ;FOLD -- Start Dress Fin AUS -- ;%{SE}%MKUKATPVW %CVW_COM %VCOMMENT %P 2:-- Start Dress Fin AUS --, 3: VW_COMMENT
      ;ENDFOLD
      ;FOLD A3936 = AUS ;%{SE}%MKUKATPVW %CVW_SPS %VBOASG %P 2:A3936 = AUS, 3: BOASG
         $OUT[3936] = FALSE
      ;ENDFOLD
      ;FOLD -- Start StartAcknowledge AUS -- ;%{SE}%MKUKATPVW %CVW_COM %VCOMMENT %P 2:-- Start StartAcknowledge AUS --, 3: VW_COMMENT
      ;ENDFOLD
      ;FOLD A3512 = AUS ;%{SE}%MKUKATPVW %CVW_SPS %VBOASG %P 2:A3512 = AUS, 3: BOASG
         $OUT[3512] = FALSE
      ;ENDFOLD
      ;FOLD -- RSK Sammelstoerung -- ;%{SE}%MKUKATPVW %CVW_COM %VCOMMENT %P 2:-- RSK Sammelstoerung --, 3: VW_COMMENT
      ;ENDFOLD
      ;FOLD F326 = EIN ;%{SE}%MKUKATPVW %CVW_SPS %VBOASG %P 2:F326 = EIN, 3: BOASG
         $FLAG[326] = TRUE
      ;ENDFOLD
      ;FOLD F329 = F326 ;%{SE}%MKUKATPVW %CVW_SPS %VBOASG %P 2:F329 = F326, 3: BOASG
         $FLAG[329] = $FLAG[326]
      ;ENDFOLD
      ;FOLD -- Flagbildung Wiederholfraesen -- ;%{SE}%MKUKATPVW %CVW_COM %VCOMMENT %P 2:-- Flagbildung Wiederholfraesen --, 3: VW_COMMENT
      ;ENDFOLD
      ;FOLD F749 = F329 & !F748 ;%{SE}%MKUKATPVW %CVW_SPS %VBOASG %P 2:F749 = F329 & !F748, 3: BOASG
         $FLAG[749] = $FLAG[329] AND NOT $FLAG[748]
      ;ENDFOLD
      ;FOLD Schritt 500 = A4039 & F329 & A3926 & (E26 + E27) ;%{SE}%MKUKATPVW %CVW_SPS %VST_CON %P 2:Schritt 500 = A4039 & F329 & A3926 & (E26 + E27), 3: ST_CON
         IF $OUT[4039] AND $FLAG[329] AND $OUT[3926] AND ($IN[26] OR $IN[27]) THEN
            PREV_STEP[9] = APP_INT_STEP[9]
            APP_INT_STEP[9] = 500
         ENDIF
      ;ENDFOLD
   ;ENDFOLD
   ;FOLD SCHRITT 505 -- rob. RZ # Acknowledge -- ;%{P}%MKUKATPVW,%CSTEP,%VST_NR,%P 1:SCHRITT, 2:505, 3: rob. RZ # Acknowledge
      ;FOLD ;%{H}
         Case 505
      ;ENDFOLD
      ;FOLD -- Ausblasen AUS -- ;%{SE}%MKUKATPVW %CVW_COM %VCOMMENT %P 2:-- Ausblasen AUS --, 3: VW_COMMENT
      ;ENDFOLD
      ;FOLD A834 = AUS ;%{SE}%MKUKATPVW %CVW_SPS %VBOASG %P 2:A834 = AUS, 3: BOASG
         $OUT[834] = FALSE
      ;ENDFOLD
      ;FOLD A835 = AUS ;%{SE}%MKUKATPVW %CVW_SPS %VBOASG %P 2:A835 = AUS, 3: BOASG
         $OUT[835] = FALSE
      ;ENDFOLD
      ;FOLD A858 = AUS ;%{SE}%MKUKATPVW %CVW_SPS %VBOASG %P 2:A858 = AUS, 3: BOASG
         $OUT[858] = FALSE
      ;ENDFOLD
      ;FOLD A859 = AUS ;%{SE}%MKUKATPVW %CVW_SPS %VBOASG %P 2:A859 = AUS, 3: BOASG
         $OUT[859] = FALSE
      ;ENDFOLD
      ;FOLD -- ServoGun - StartAcknowledge -- ;%{SE}%MKUKATPVW %CVW_COM %VCOMMENT %P 2:-- ServoGun - StartAcknowledge --, 3: VW_COMMENT
      ;ENDFOLD
      ;FOLD A3510 = AUS ;%{SE}%MKUKATPVW %CVW_SPS %VBOASG %P 2:A3510 = AUS, 3: BOASG
         $OUT[3510] = FALSE
      ;ENDFOLD
      ;FOLD A3514 = AUS ;%{SE}%MKUKATPVW %CVW_SPS %VBOASG %P 2:A3514 = AUS, 3: BOASG
         $OUT[3514] = FALSE
      ;ENDFOLD
      ;FOLD A3512 = EIN ;%{SE}%MKUKATPVW %CVW_SPS %VBOASG %P 2:A3512 = EIN, 3: BOASG
         $OUT[3512] = TRUE
      ;ENDFOLD
      ;FOLD Schritt 506 = !F335 & A4039 & !A3507 ;%{SE}%MKUKATPVW %CVW_SPS %VST_CON %P 2:Schritt 506 = !F335 & A4039 & !A3507, 3: ST_CON
         IF NOT $FLAG[335] AND $OUT[4039] AND NOT $OUT[3507] THEN
            PREV_STEP[9] = APP_INT_STEP[9]
            APP_INT_STEP[9] = 506
         ENDIF
      ;ENDFOLD
      ;FOLD Schritt 506 = F335 & !F78 & A4039 & !A3507 ;%{SE}%MKUKATPVW %CVW_SPS %VST_CON %P 2:Schritt 506 = F335 & !F78 & A4039 & !A3507, 3: ST_CON
         IF $FLAG[335] AND NOT $FLAG[78] AND $OUT[4039] AND NOT $OUT[3507] THEN
            PREV_STEP[9] = APP_INT_STEP[9]
            APP_INT_STEP[9] = 506
         ENDIF
      ;ENDFOLD
   ;ENDFOLD
   ;FOLD SCHRITT 506 -- rob. RZ # Ruecksetzen -- ;%{P}%MKUKATPVW,%CSTEP,%VST_NR,%P 1:SCHRITT, 2:506, 3: rob. RZ # Ruecksetzen
      ;FOLD ;%{H}
         Case 506
      ;ENDFOLD
      ;FOLD -- Start Init Same AUS -- ;%{SE}%MKUKATPVW %CVW_COM %VCOMMENT %P 2:-- Start Init Same AUS --, 3: VW_COMMENT
      ;ENDFOLD
      ;FOLD A3514 = AUS ;%{SE}%MKUKATPVW %CVW_SPS %VBOASG %P 2:A3514 = AUS, 3: BOASG
         $OUT[3514] = FALSE
      ;ENDFOLD
      ;FOLD -- Start Spot AUS -- ;%{SE}%MKUKATPVW %CVW_COM %VCOMMENT %P 2:-- Start Spot AUS --, 3: VW_COMMENT
      ;ENDFOLD
      ;FOLD A3511 = AUS ;%{SE}%MKUKATPVW %CVW_SPS %VBOASG %P 2:A3511 = AUS, 3: BOASG
         $OUT[3511] = FALSE
      ;ENDFOLD
      ;FOLD -- Start Dress AUS -- ;%{SE}%MKUKATPVW %CVW_COM %VCOMMENT %P 2:-- Start Dress AUS --, 3: VW_COMMENT
      ;ENDFOLD
      ;FOLD A3510 = AUS ;%{SE}%MKUKATPVW %CVW_SPS %VBOASG %P 2:A3510 = AUS, 3: BOASG
         $OUT[3510] = FALSE
      ;ENDFOLD
      ;FOLD -- Start Init New AUS -- ;%{SE}%MKUKATPVW %CVW_COM %VCOMMENT %P 2:-- Start Init New AUS --, 3: VW_COMMENT
      ;ENDFOLD
      ;FOLD A3513 = AUS ;%{SE}%MKUKATPVW %CVW_SPS %VBOASG %P 2:A3513 = AUS, 3: BOASG
         $OUT[3513] = FALSE
      ;ENDFOLD
      ;FOLD -- Start Dress in Position AUS -- ;%{SE}%MKUKATPVW %CVW_COM %VCOMMENT %P 2:-- Start Dress in Position AUS --, 3: VW_COMMENT
      ;ENDFOLD
      ;FOLD A3935 = AUS ;%{SE}%MKUKATPVW %CVW_SPS %VBOASG %P 2:A3935 = AUS, 3: BOASG
         $OUT[3935] = FALSE
      ;ENDFOLD
      ;FOLD -- Start Dress Fin AUS -- ;%{SE}%MKUKATPVW %CVW_COM %VCOMMENT %P 2:-- Start Dress Fin AUS --, 3: VW_COMMENT
      ;ENDFOLD
      ;FOLD A3936 = AUS ;%{SE}%MKUKATPVW %CVW_SPS %VBOASG %P 2:A3936 = AUS, 3: BOASG
         $OUT[3936] = FALSE
      ;ENDFOLD
      ;FOLD -- Start StartAcknowledge AUS -- ;%{SE}%MKUKATPVW %CVW_COM %VCOMMENT %P 2:-- Start StartAcknowledge AUS --, 3: VW_COMMENT
      ;ENDFOLD
      ;FOLD A3512 = AUS ;%{SE}%MKUKATPVW %CVW_SPS %VBOASG %P 2:A3512 = AUS, 3: BOASG
         $OUT[3512] = FALSE
      ;ENDFOLD
      ;FOLD -- Fehler SK ruecksetzen -- ;%{SE}%MKUKATPVW %CVW_COM %VCOMMENT %P 2:-- Fehler SK ruecksetzen --, 3: VW_COMMENT
      ;ENDFOLD
      ;FOLD -- Druckvorgabe SK1/ServoGun -- ;%{SE}%MKUKATPVW %CVW_COM %VCOMMENT %P 2:-- Druckvorgabe SK1/ServoGun --, 3: VW_COMMENT
      ;ENDFOLD
      ;FOLD bin1 ( F78 ) = 41 ;%{SE}%MKUKATPVW %CVW_SPS %VARIASG %P 2:bin1 ( F78 ) = 41, 3: ARIASG
         VW(#BINOUT,$FLAG[78],1,41)
      ;ENDFOLD
      ;FOLD bin1 ( F79 ) = 51 ;%{SE}%MKUKATPVW %CVW_SPS %VARIASG %P 2:bin1 ( F79 ) = 51, 3: ARIASG
         VW(#BINOUT,$FLAG[79],1,51)
      ;ENDFOLD
      ;FOLD bin31 ( F78 ) = 41 ;%{SE}%MKUKATPVW %CVW_SPS %VARIASG %P 2:bin31 ( F78 ) = 41, 3: ARIASG
         VW(#BINOUT,$FLAG[78],31,41)
      ;ENDFOLD
      ;FOLD bin31 ( F79 ) = 51 ;%{SE}%MKUKATPVW %CVW_SPS %VARIASG %P 2:bin31 ( F79 ) = 51, 3: ARIASG
         VW(#BINOUT,$FLAG[79],31,51)
      ;ENDFOLD
      ;FOLD -- Wartezeit Programmwechsel SK -- ;%{SE}%MKUKATPVW %CVW_COM %VCOMMENT %P 2:-- Wartezeit Programmwechsel SK --, 3: VW_COMMENT
      ;ENDFOLD
      ;FOLD T8 ( !F334 ) = -2[1/10Sek] ;%{SE}%MKUKATPVW %CVW_SPS %VTASG %P 2:T8 ( !F334 ) = -2[1/10Sek], 3: TASG
         VW(#SET_TIME,NOT $FLAG[334],8,0,-2)
      ;ENDFOLD
      ;FOLD -- Hilfsflag SK Programmwechsel -- ;%{SE}%MKUKATPVW %CVW_COM %VCOMMENT %P 2:-- Hilfsflag SK Programmwechsel --, 3: VW_COMMENT
      ;ENDFOLD
      ;FOLD F334 = EIN ;%{SE}%MKUKATPVW %CVW_SPS %VBOASG %P 2:F334 = EIN, 3: BOASG
         $FLAG[334] = TRUE
      ;ENDFOLD
      ;FOLD t9 ( EIN ) = STOP ;%{SE}%MKUKATPVW %CVW_SPS %VTSTOP %P 2:t9 ( EIN ) = STOP, 3: TSTOP
         VW(#SET_TIME,TRUE,9,1,0)
      ;ENDFOLD
      ;FOLD Schritt 1 = T8 & A4039 & A3506 & A3505 ;%{SE}%MKUKATPVW %CVW_SPS %VST_CON %P 2:Schritt 1 = T8 & A4039 & A3506 & A3505, 3: ST_CON
         IF $TIMER_FLAG[8] AND $OUT[4039] AND $OUT[3506] AND $OUT[3505] THEN
            PREV_STEP[9] = APP_INT_STEP[9]
            APP_INT_STEP[9] = 1
         ENDIF
      ;ENDFOLD
   ;ENDFOLD
   ; FOLD ;%{H}
   DEFAULT
   HMeldung ("StepNotAvailableInModul")
   APP_INT_STEP[9]=1
   ENDSWITCH
   END
   DEF HMeldung (Meld[]:IN)
     CHAR Meld[]
     DECL KrlMsg_T Msg
     DECL KrlMsgPar_T Par[3]
     DECL KrlMsgOpt_T Opt
     INT nHandle
     BOOL dummy
     dummy=STRCOPY(Msg.Msg_txt[],Meld[])
     Msg.Modul[]="MAKROSTEP"
     Msg.Nr=111
     Par[1].Par_type=#Value
     Par[1].Par_Txt[] = "9"
     Par[2].Par_type=#Value
     Par[2].Par_Int = PREV_STEP[9]
     Opt = {VL_Stop TRUE, Clear_P_Reset TRUE, Log_To_DB FALSE}
     nHandle = Set_KrlMsg (#Notify, Msg, Par[], Opt)
     WAIT SEC 0.2
END
; ENDFOLD
